# EPICS IOC start-up script: iocsh/EthercatMCAxisdebug.iocsh
dbLoadRecords("EthercatMCdebug.template", "PREFIX=$(PREFIX), MOTOR_NAME=$(MOTOR_NAME), MOTOR_PORT=$(MOTOR_PORT), AXIS_NO=$(AXIS_NO), PREC=3")
